(* Logix 5000 project; controller HP_SSC01 vendor 1 type 14 code 67 rev 17.7; software revision 17.01; part 9 of 15 *)
(* tags used below, declared in another part *)
   A_C3_0218 : ALIAS FOR S_C3_FaultSafety.18;
   A_C3_0219 : ALIAS FOR S_C3_FaultSafety.19;
   A_C3_0220 : ALIAS FOR S_C3_FaultSafety.20;
   A_C3_0221 : ALIAS FOR S_C3_FaultSafety.21;
   A_C3_0222 : ALIAS FOR S_C3_FaultSafety.22;
   A_C3_0223 : ALIAS FOR S_C3_FaultSafety.23;
   A_C3_0311 : ALIAS FOR C3_FaultStandard.11;
   A_C3_0312 : ALIAS FOR C3_FaultStandard.12;
   A_C3_0313 : ALIAS FOR C3_FaultStandard.13;
   A_C3_0314 : ALIAS FOR C3_FaultStandard.14;
   A_C3_0315 : ALIAS FOR C3_FaultStandard.15;
   C3 : AXIS_SERVO_DRIVE;
   C3_EncoderDegree : REAL;
   C3_EncoderPositionAtHome : DINT;
   C3_ExcecutePBHoldTimer : TIMER;
   C3_FaultHomeSwitchNotFound : BOOL;
   C3_Homed : BOOL;
   C3_HomeDelay : TIMER[8];
   C3_HomeFindSwitchMAM01 : MOTION_INSTRUCTION;
   C3_HomeFindSwitchMAM02 : MOTION_INSTRUCTION;
   C3_HomeFindSwitchMAS01 : MOTION_INSTRUCTION;
   C3_HomeGetCloseToSwitchMAM01 : MOTION_INSTRUCTION;
   C3_HomeGoToOnPathMAM01 : MOTION_INSTRUCTION;
   C3_HomeMessageNumber : DINT;
   C3_HomeSensorTestMAM02 : MOTION_INSTRUCTION;
   C3_HomeSequence : DINT;
   C3_HomeSequenceAlarms : DINT;
   C3_HomeSequenceAlarmTimer : TIMER[32];
   C3_HomeSequenceInProcess : BOOL;
   C3_HomeSequenceMAH : MOTION_INSTRUCTION;
   C3_HomeSwitchFaultK7KFailedOff : BOOL;
   C3_HomeSwitchFaultK7KFailedOn : BOOL;
   C3_HomeSwitchFaultSafeFailedOff : BOOL;
   C3_HomeSwitchFaultSafeFailedOn : BOOL;
   C3_HomeTest : REAL;
   C3_IndexEnable : BOOL;
   C3_IndexEnableTOF : TIMER;
   C3_IndexMAM01 : MOTION_INSTRUCTION;
   C3_IndexMAS01 : MOTION_INSTRUCTION;
   C3_IndexMessageNumber : DINT;
   C3_IndexPermissive : BOOL;
   C3_Jog_ONS : DINT;
   C3_JogDirection : DINT;
   C3_JogEnable : BOOL;
   C3_JogEnableTOF : TIMER;
   C3_JogForwardFastSelected : BOOL;
   C3_JogForwardSlowSelected : BOOL;
   C3_JogMAJ01 : MOTION_INSTRUCTION;
   C3_JogMAJ02 : MOTION_INSTRUCTION;
   C3_JogMAS01 : MOTION_INSTRUCTION;
   C3_JogMessageNumber : DINT;
   C3_JogPermissive : BOOL;
   C3_JogReverseFastSelected : BOOL;
   C3_JogReverseSlowSelected : BOOL;
   C3_MAJAcceleration : REAL;
   C3_MAJDeceleration : REAL;
   C3_MAJSpeed : REAL;
   C3_OIT_Current : DINT;
   C3_RemoteHomeCMD : BOOL;
   C3_ServoActionStatusOnDelay : TIMER;
   C3_SetEncoderHomePosition : BOOL;
   C3HomeSensorTestMAM01 : MOTION_INSTRUCTION;
   C3HomeSequenceONS : BOOL;
   C3HomeSequenceONS2 : BOOL;
   S_C3_EncoderPositionAtHomeSet : BOOL;
   S_C3_ExecutePB : BOOL;
   S_C3_FaultReset : BOOL;
   S_C3_HomeSafePE : ALIAS FOR C3_Safe:I.Pt04Data;
   S_C3_ModeLocal : BOOL;
   S_C3_ModeRemote : BOOL;
   S_C3_MSTOP_InputOK : BOOL;
   S_EncoderCtsFor360Deg : DINT;
(* Carousel3, continued *)

ROUTINE C330_Home   (* ladder *)
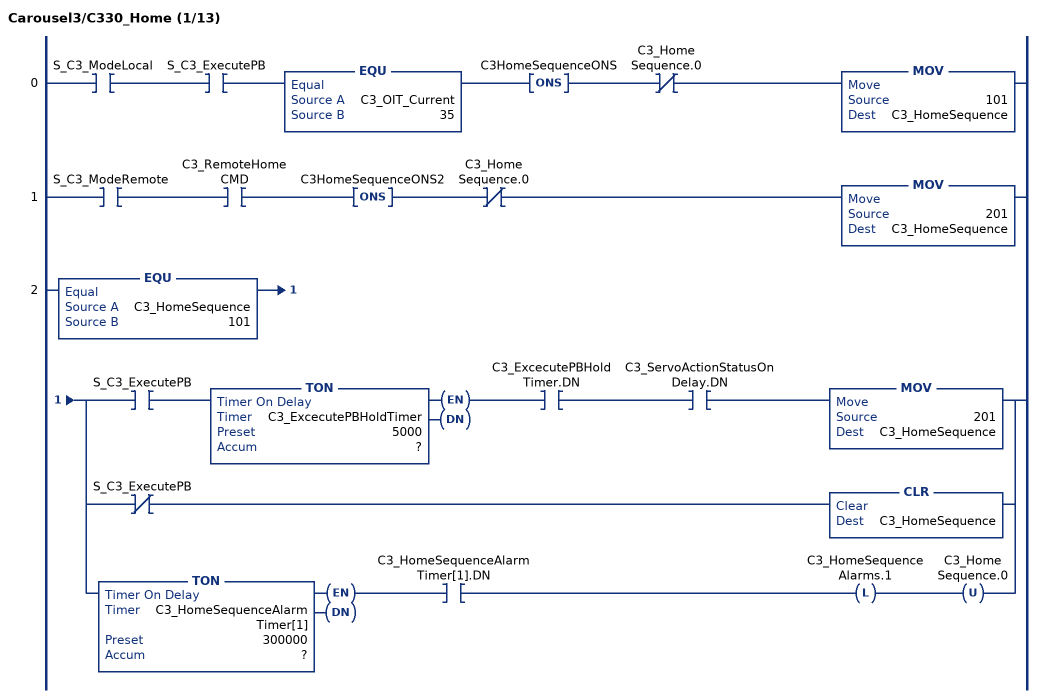
   0: XIC(S_C3_ModeLocal)XIC(S_C3_ExecutePB)EQU(C3_OIT_Current,35)ONS(C3HomeSequenceONS)XIO(C3_HomeSequence.0)MOV(101,C3_HomeSequence);
   1: XIC(S_C3_ModeRemote)XIC(C3_RemoteHomeCMD)ONS(C3HomeSequenceONS2)XIO(C3_HomeSequence.0)MOV(201,C3_HomeSequence);
   2: EQU(C3_HomeSequence,101)[XIC(S_C3_ExecutePB) TON(C3_ExcecutePBHoldTimer,?,?) XIC(C3_ExcecutePBHoldTimer.DN) XIC(C3_ServoActionStatusOnDelay.DN) MOV(201,C3_HomeSequence) ,XIO(S_C3_ExecutePB) CLR(C3_HomeSequence) ,TON(C3_HomeSequenceAlarmTimer[1],?,?) XIC(C3_HomeSequenceAlarmTimer[1].DN) OTL(C3_HomeSequenceAlarms.1) OTU(C3_HomeSequence.0) ];
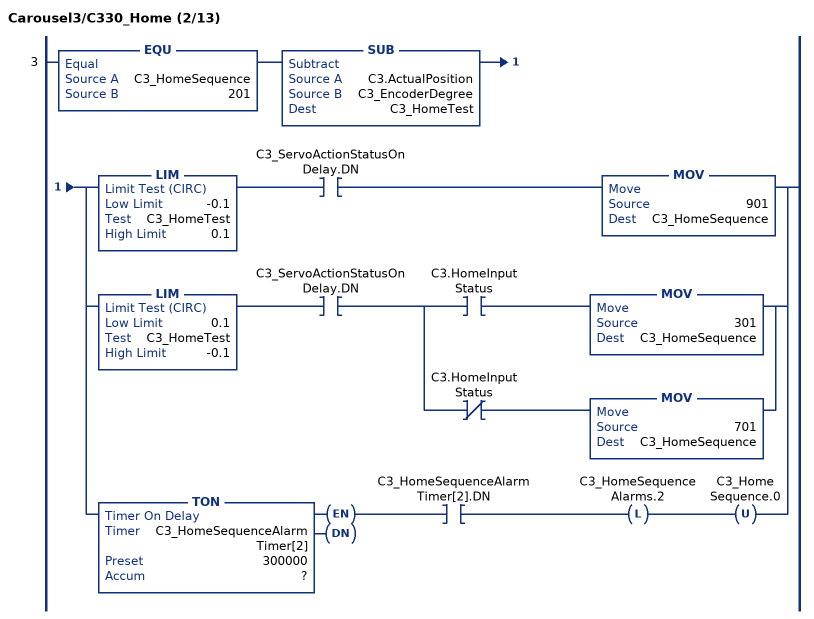
   3: EQU(C3_HomeSequence,201)SUB(C3.ActualPosition,C3_EncoderDegree,C3_HomeTest)[LIM(-0.1,C3_HomeTest,0.1) XIC(C3_ServoActionStatusOnDelay.DN) MOV(901,C3_HomeSequence) ,LIM(0.1,C3_HomeTest,-0.1) XIC(C3_ServoActionStatusOnDelay.DN) [XIC(C3.HomeInputStatus) MOV(301,C3_HomeSequence) ,XIO(C3.HomeInputStatus) MOV(701,C3_HomeSequence) ] ,TON(C3_HomeSequenceAlarmTimer[2],?,?) XIC(C3_HomeSequenceAlarmTimer[2].DN) OTL(C3_HomeSequenceAlarms.2) OTU(C3_HomeSequence.0) ];
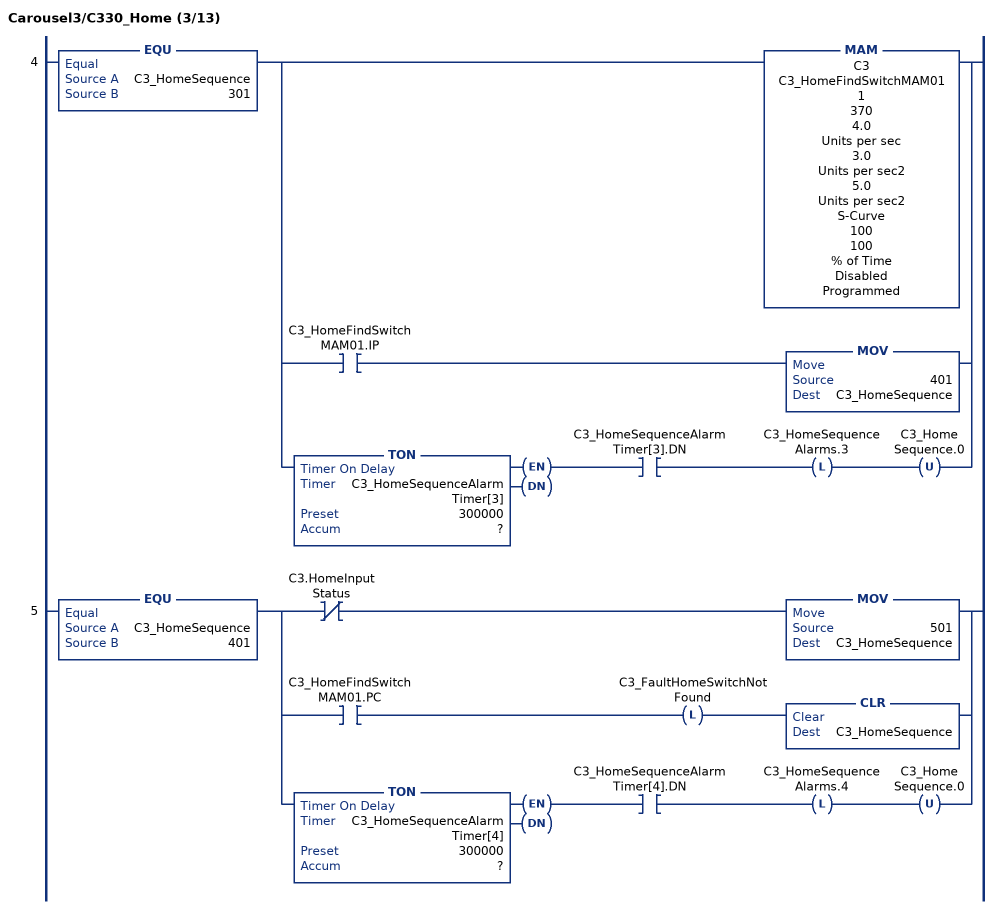
   4: EQU(C3_HomeSequence,301)[MAM(C3,C3_HomeFindSwitchMAM01,1,370,4.0,Units per sec,3.0,Units per sec2,5.0,Units per sec2,S-Curve,100,100,% of Time,Disabled,Programmed) ,XIC(C3_HomeFindSwitchMAM01.IP) MOV(401,C3_HomeSequence) ,TON(C3_HomeSequenceAlarmTimer[3],?,?) XIC(C3_HomeSequenceAlarmTimer[3].DN) OTL(C3_HomeSequenceAlarms.3) OTU(C3_HomeSequence.0) ];
   5: EQU(C3_HomeSequence,401)[XIO(C3.HomeInputStatus) MOV(501,C3_HomeSequence) ,XIC(C3_HomeFindSwitchMAM01.PC) OTL(C3_FaultHomeSwitchNotFound) CLR(C3_HomeSequence) ,TON(C3_HomeSequenceAlarmTimer[4],?,?) XIC(C3_HomeSequenceAlarmTimer[4].DN) OTL(C3_HomeSequenceAlarms.4) OTU(C3_HomeSequence.0) ];
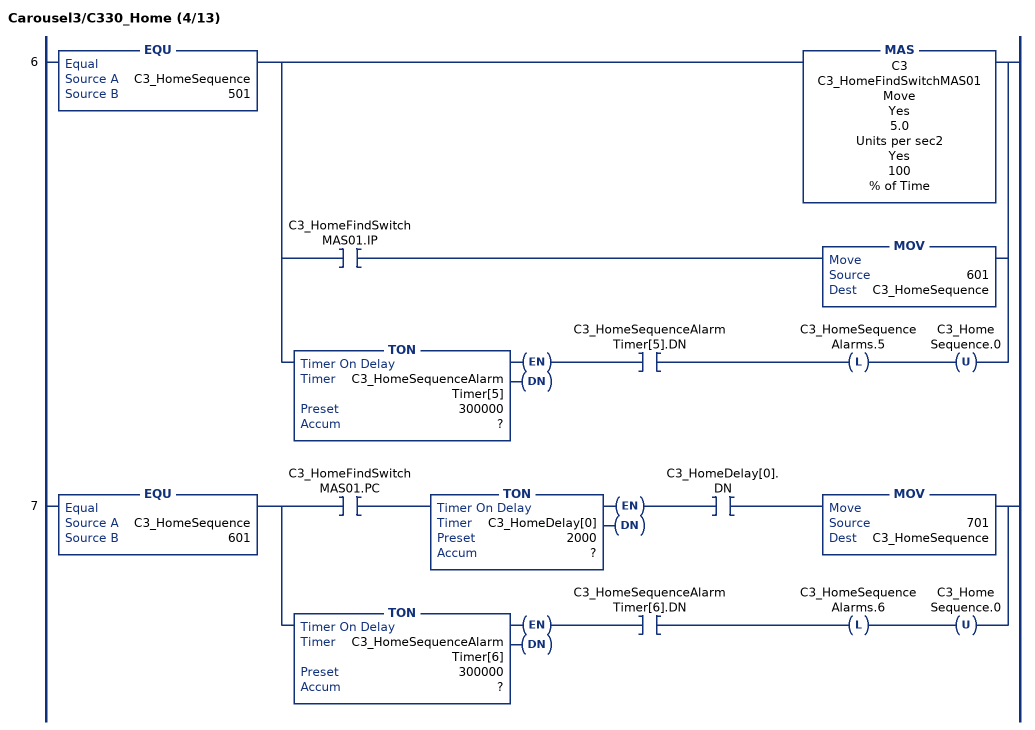
   6: EQU(C3_HomeSequence,501)[MAS(C3,C3_HomeFindSwitchMAS01,Move,Yes,5.0,Units per sec2,Yes,100,% of Time) ,XIC(C3_HomeFindSwitchMAS01.IP) MOV(601,C3_HomeSequence) ,TON(C3_HomeSequenceAlarmTimer[5],?,?) XIC(C3_HomeSequenceAlarmTimer[5].DN) OTL(C3_HomeSequenceAlarms.5) OTU(C3_HomeSequence.0) ];
   7: EQU(C3_HomeSequence,601)[XIC(C3_HomeFindSwitchMAS01.PC) TON(C3_HomeDelay[0],?,?) XIC(C3_HomeDelay[0].DN) MOV(701,C3_HomeSequence) ,TON(C3_HomeSequenceAlarmTimer[6],?,?) XIC(C3_HomeSequenceAlarmTimer[6].DN) OTL(C3_HomeSequenceAlarms.6) OTU(C3_HomeSequence.0) ];
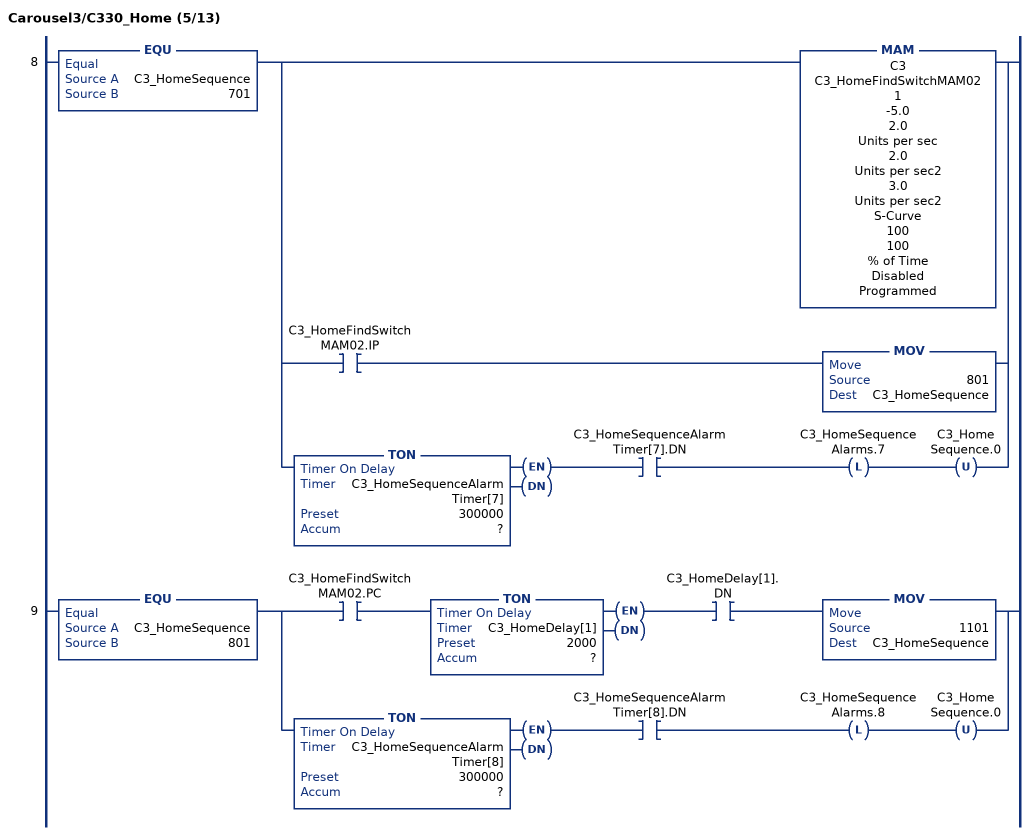
   8: EQU(C3_HomeSequence,701)[MAM(C3,C3_HomeFindSwitchMAM02,1,-5.0,2.0,Units per sec,2.0,Units per sec2,3.0,Units per sec2,S-Curve,100,100,% of Time,Disabled,Programmed) ,XIC(C3_HomeFindSwitchMAM02.IP) MOV(801,C3_HomeSequence) ,TON(C3_HomeSequenceAlarmTimer[7],?,?) XIC(C3_HomeSequenceAlarmTimer[7].DN) OTL(C3_HomeSequenceAlarms.7) OTU(C3_HomeSequence.0) ];
   9: EQU(C3_HomeSequence,801)[XIC(C3_HomeFindSwitchMAM02.PC) TON(C3_HomeDelay[1],?,?) XIC(C3_HomeDelay[1].DN) MOV(1101,C3_HomeSequence) ,TON(C3_HomeSequenceAlarmTimer[8],?,?) XIC(C3_HomeSequenceAlarmTimer[8].DN) OTL(C3_HomeSequenceAlarms.8) OTU(C3_HomeSequence.0) ];
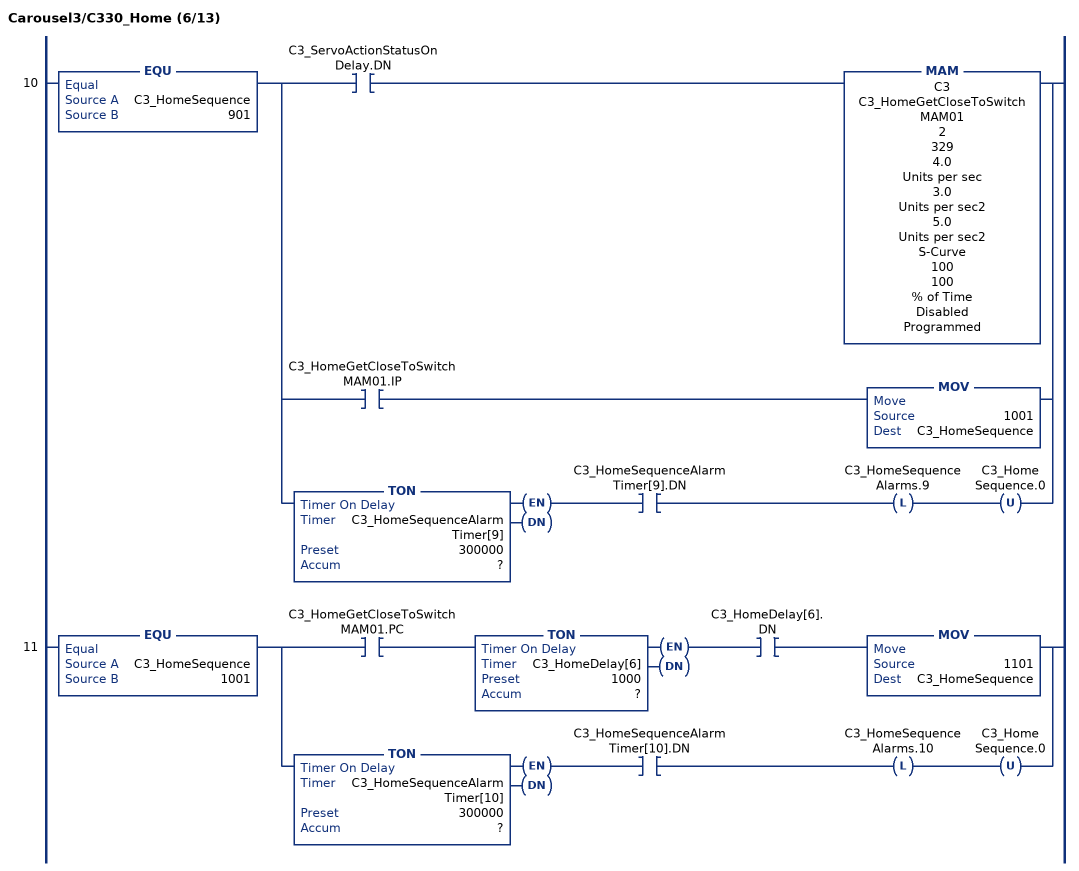
   10: EQU(C3_HomeSequence,901)[XIC(C3_ServoActionStatusOnDelay.DN) MAM(C3,C3_HomeGetCloseToSwitchMAM01,2,329,4.0,Units per sec,3.0,Units per sec2,5.0,Units per sec2,S-Curve,100,100,% of Time,Disabled,Programmed) ,XIC(C3_HomeGetCloseToSwitchMAM01.IP) MOV(1001,C3_HomeSequence) ,TON(C3_HomeSequenceAlarmTimer[9],?,?) XIC(C3_HomeSequenceAlarmTimer[9].DN) OTL(C3_HomeSequenceAlarms.9) OTU(C3_HomeSequence.0) ];
   11: EQU(C3_HomeSequence,1001)[XIC(C3_HomeGetCloseToSwitchMAM01.PC) TON(C3_HomeDelay[6],?,?) XIC(C3_HomeDelay[6].DN) MOV(1101,C3_HomeSequence) ,TON(C3_HomeSequenceAlarmTimer[10],?,?) XIC(C3_HomeSequenceAlarmTimer[10].DN) OTL(C3_HomeSequenceAlarms.10) OTU(C3_HomeSequence.0) ];
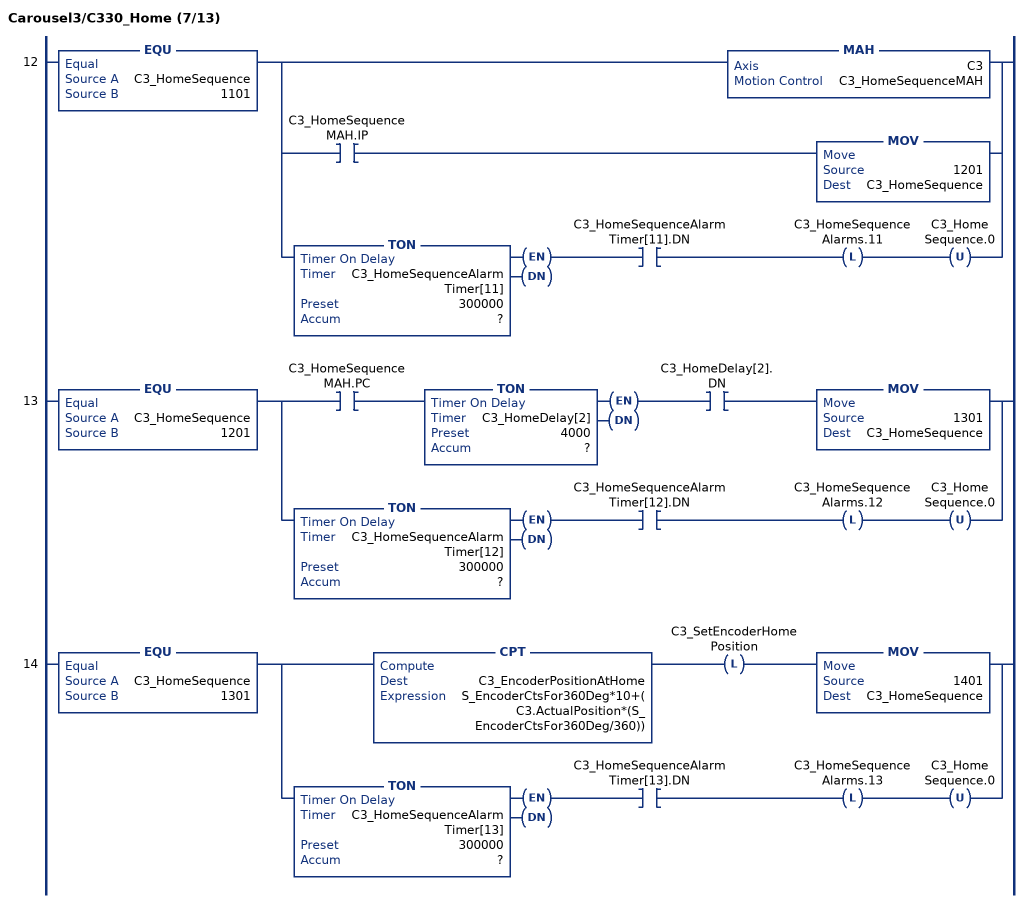
   12: EQU(C3_HomeSequence,1101)[MAH(C3,C3_HomeSequenceMAH) ,XIC(C3_HomeSequenceMAH.IP) MOV(1201,C3_HomeSequence) ,TON(C3_HomeSequenceAlarmTimer[11],?,?) XIC(C3_HomeSequenceAlarmTimer[11].DN) OTL(C3_HomeSequenceAlarms.11) OTU(C3_HomeSequence.0) ];
   13: EQU(C3_HomeSequence,1201)[XIC(C3_HomeSequenceMAH.PC) TON(C3_HomeDelay[2],?,?) XIC(C3_HomeDelay[2].DN) MOV(1301,C3_HomeSequence) ,TON(C3_HomeSequenceAlarmTimer[12],?,?) XIC(C3_HomeSequenceAlarmTimer[12].DN) OTL(C3_HomeSequenceAlarms.12) OTU(C3_HomeSequence.0) ];
   14: EQU(C3_HomeSequence,1301)[CPT(C3_EncoderPositionAtHome,S_EncoderCtsFor360Deg*10+(C3.ActualPosition*(S_EncoderCtsFor360Deg/360))) OTL(C3_SetEncoderHomePosition) MOV(1401,C3_HomeSequence) ,TON(C3_HomeSequenceAlarmTimer[13],?,?) XIC(C3_HomeSequenceAlarmTimer[13].DN) OTL(C3_HomeSequenceAlarms.13) OTU(C3_HomeSequence.0) ];
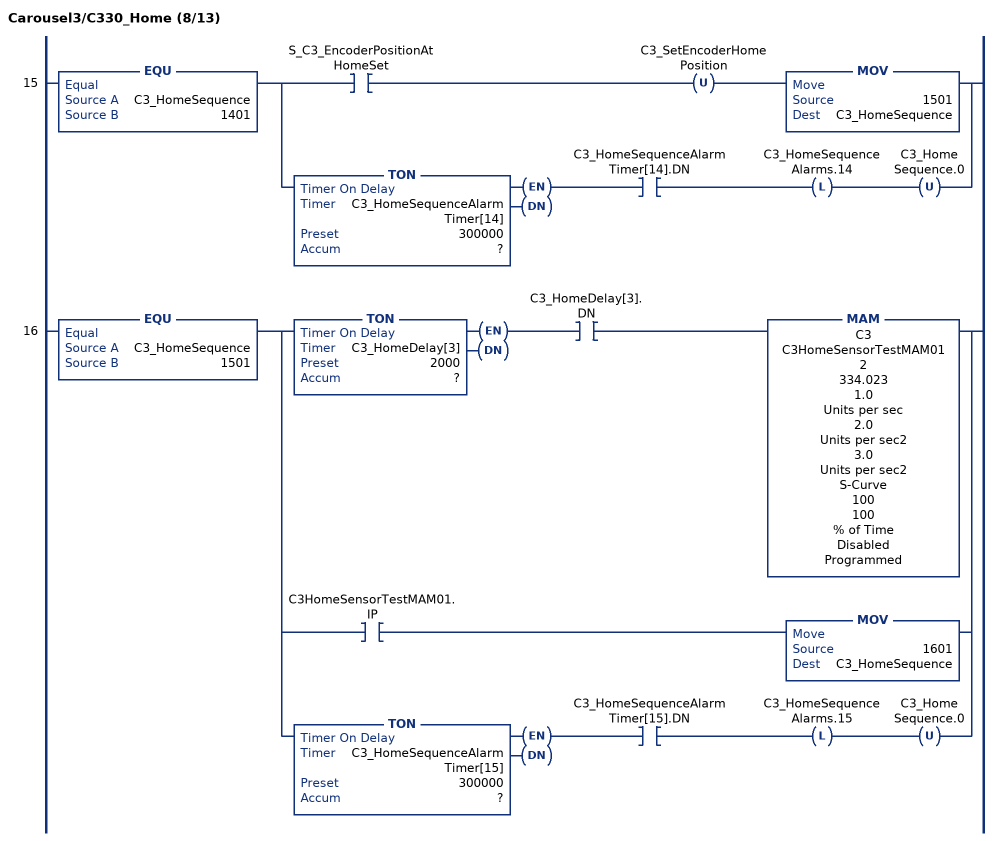
   15: EQU(C3_HomeSequence,1401)[XIC(S_C3_EncoderPositionAtHomeSet) OTU(C3_SetEncoderHomePosition) MOV(1501,C3_HomeSequence) ,TON(C3_HomeSequenceAlarmTimer[14],?,?) XIC(C3_HomeSequenceAlarmTimer[14].DN) OTL(C3_HomeSequenceAlarms.14) OTU(C3_HomeSequence.0) ];
   16: EQU(C3_HomeSequence,1501)[TON(C3_HomeDelay[3],?,?) XIC(C3_HomeDelay[3].DN) MAM(C3,C3HomeSensorTestMAM01,2,334.023,1.0,Units per sec,2.0,Units per sec2,3.0,Units per sec2,S-Curve,100,100,% of Time,Disabled,Programmed) ,XIC(C3HomeSensorTestMAM01.IP) MOV(1601,C3_HomeSequence) ,TON(C3_HomeSequenceAlarmTimer[15],?,?) XIC(C3_HomeSequenceAlarmTimer[15].DN) OTL(C3_HomeSequenceAlarms.15) OTU(C3_HomeSequence.0) ];
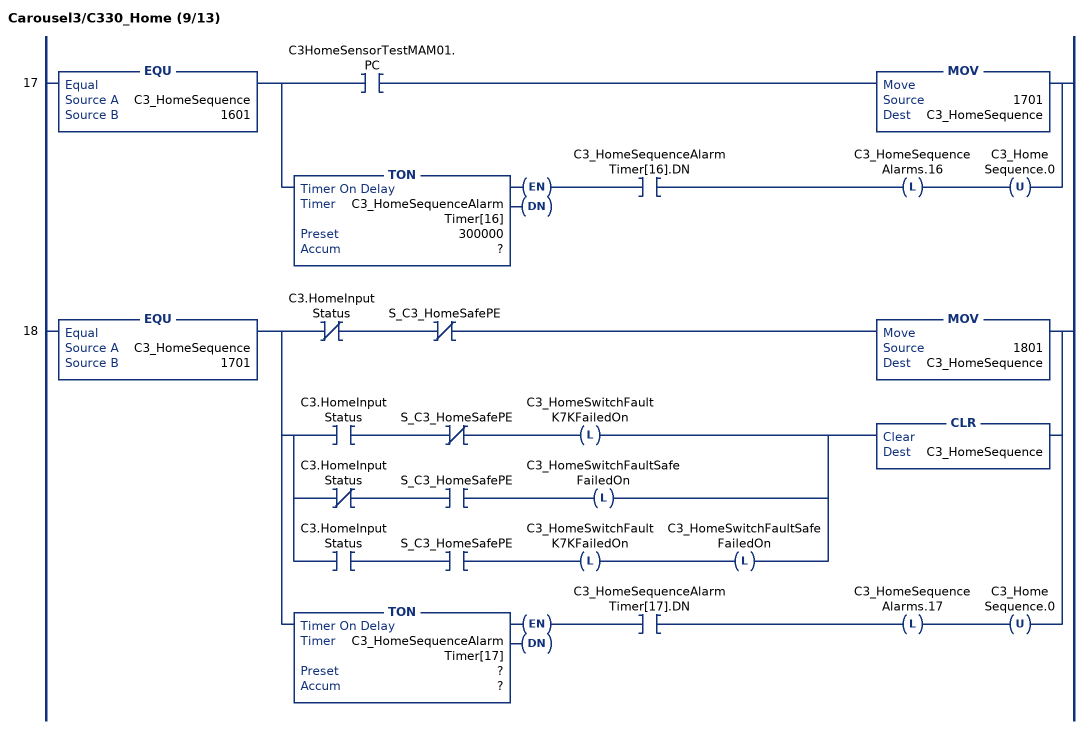
   17: EQU(C3_HomeSequence,1601)[XIC(C3HomeSensorTestMAM01.PC) MOV(1701,C3_HomeSequence) ,TON(C3_HomeSequenceAlarmTimer[16],?,?) XIC(C3_HomeSequenceAlarmTimer[16].DN) OTL(C3_HomeSequenceAlarms.16) OTU(C3_HomeSequence.0) ];
   18: EQU(C3_HomeSequence,1701)[XIO(C3.HomeInputStatus) XIO(S_C3_HomeSafePE) MOV(1801,C3_HomeSequence) ,[XIC(C3.HomeInputStatus) XIO(S_C3_HomeSafePE) OTL(C3_HomeSwitchFaultK7KFailedOn) ,XIO(C3.HomeInputStatus) XIC(S_C3_HomeSafePE) OTL(C3_HomeSwitchFaultSafeFailedOn) ,XIC(C3.HomeInputStatus) XIC(S_C3_HomeSafePE) OTL(C3_HomeSwitchFaultK7KFailedOn) OTL(C3_HomeSwitchFaultSafeFailedOn) ] CLR(C3_HomeSequence) ,TON(C3_HomeSequenceAlarmTimer[17],?,?) XIC(C3_HomeSequenceAlarmTimer[17].DN) OTL(C3_HomeSequenceAlarms.17) OTU(C3_HomeSequence.0) ];
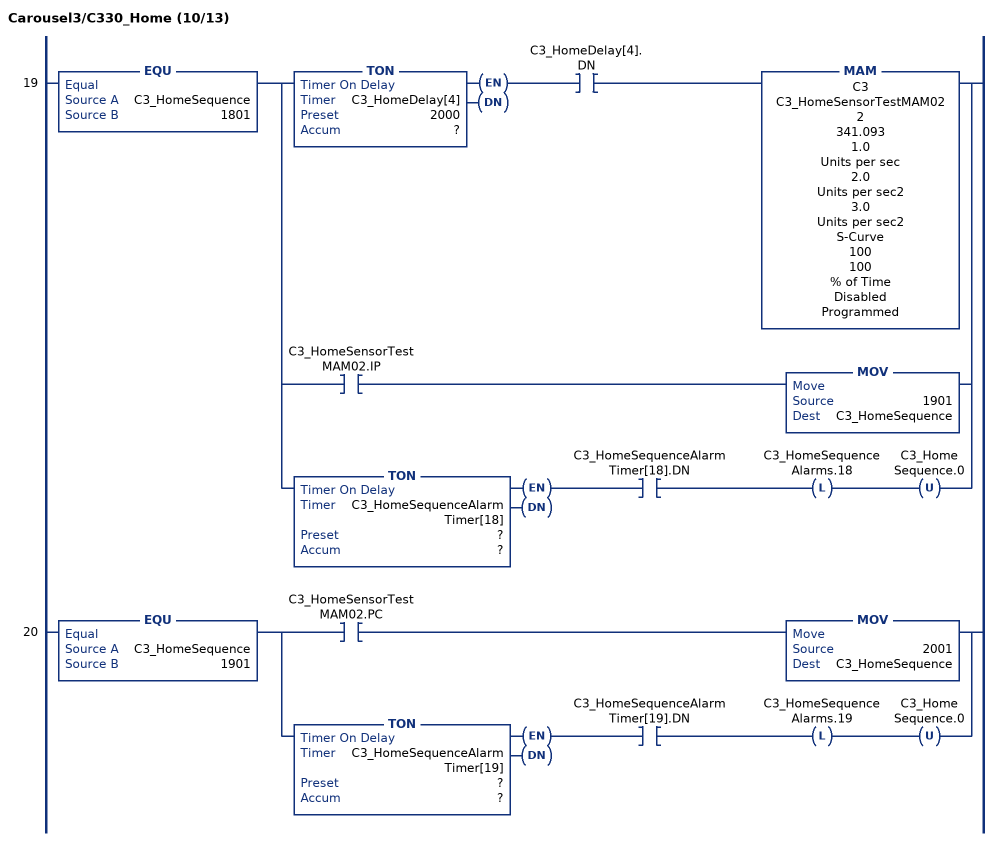
   19: EQU(C3_HomeSequence,1801)[TON(C3_HomeDelay[4],?,?) XIC(C3_HomeDelay[4].DN) MAM(C3,C3_HomeSensorTestMAM02,2,341.093,1.0,Units per sec,2.0,Units per sec2,3.0,Units per sec2,S-Curve,100,100,% of Time,Disabled,Programmed) ,XIC(C3_HomeSensorTestMAM02.IP) MOV(1901,C3_HomeSequence) ,TON(C3_HomeSequenceAlarmTimer[18],?,?) XIC(C3_HomeSequenceAlarmTimer[18].DN) OTL(C3_HomeSequenceAlarms.18) OTU(C3_HomeSequence.0) ];
   20: EQU(C3_HomeSequence,1901)[XIC(C3_HomeSensorTestMAM02.PC) MOV(2001,C3_HomeSequence) ,TON(C3_HomeSequenceAlarmTimer[19],?,?) XIC(C3_HomeSequenceAlarmTimer[19].DN) OTL(C3_HomeSequenceAlarms.19) OTU(C3_HomeSequence.0) ];
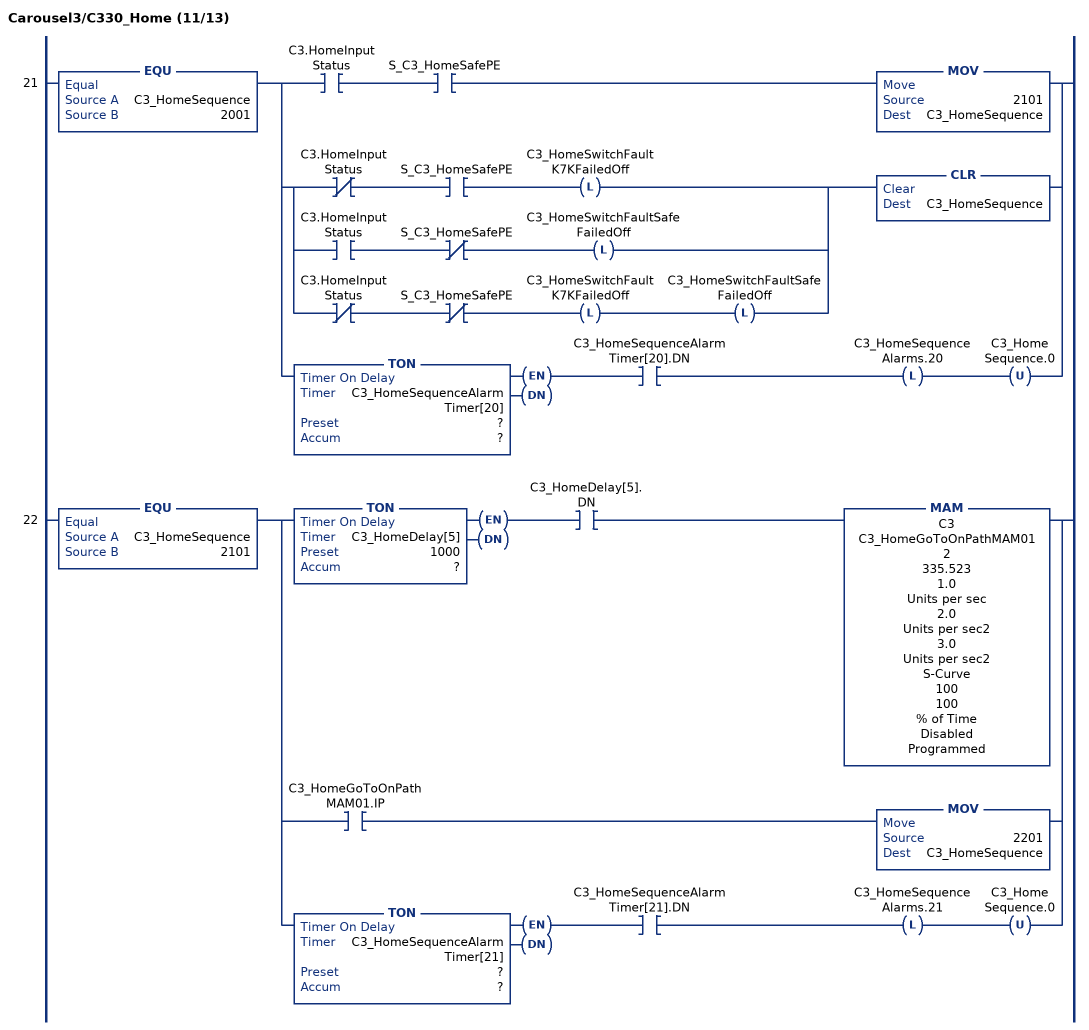
   21: EQU(C3_HomeSequence,2001)[XIC(C3.HomeInputStatus) XIC(S_C3_HomeSafePE) MOV(2101,C3_HomeSequence) ,[XIO(C3.HomeInputStatus) XIC(S_C3_HomeSafePE) OTL(C3_HomeSwitchFaultK7KFailedOff) ,XIC(C3.HomeInputStatus) XIO(S_C3_HomeSafePE) OTL(C3_HomeSwitchFaultSafeFailedOff) ,XIO(C3.HomeInputStatus) XIO(S_C3_HomeSafePE) OTL(C3_HomeSwitchFaultK7KFailedOff) OTL(C3_HomeSwitchFaultSafeFailedOff) ] CLR(C3_HomeSequence) ,TON(C3_HomeSequenceAlarmTimer[20],?,?) XIC(C3_HomeSequenceAlarmTimer[20].DN) OTL(C3_HomeSequenceAlarms.20) OTU(C3_HomeSequence.0) ];
   22: EQU(C3_HomeSequence,2101)[TON(C3_HomeDelay[5],?,?) XIC(C3_HomeDelay[5].DN) MAM(C3,C3_HomeGoToOnPathMAM01,2,335.523,1.0,Units per sec,2.0,Units per sec2,3.0,Units per sec2,S-Curve,100,100,% of Time,Disabled,Programmed) ,XIC(C3_HomeGoToOnPathMAM01.IP) MOV(2201,C3_HomeSequence) ,TON(C3_HomeSequenceAlarmTimer[21],?,?) XIC(C3_HomeSequenceAlarmTimer[21].DN) OTL(C3_HomeSequenceAlarms.21) OTU(C3_HomeSequence.0) ];
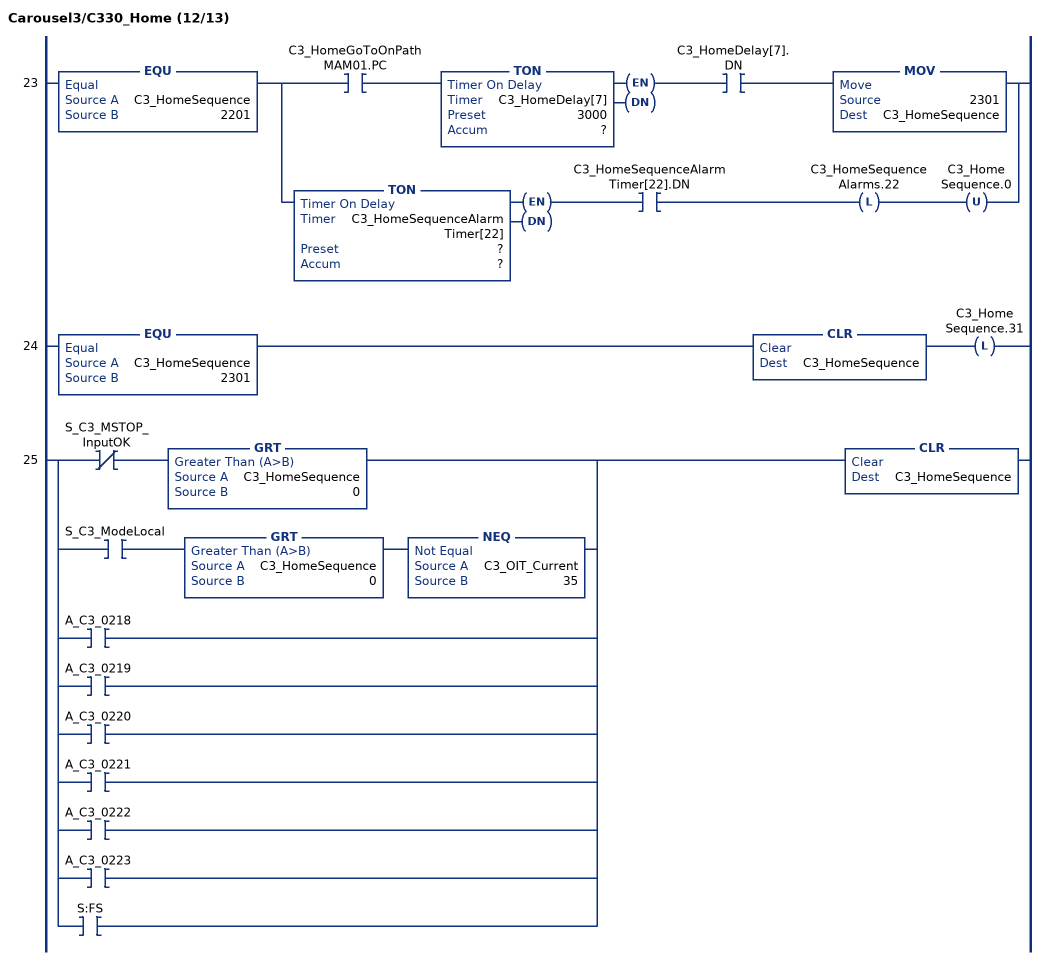
   23: EQU(C3_HomeSequence,2201)[XIC(C3_HomeGoToOnPathMAM01.PC) TON(C3_HomeDelay[7],?,?) XIC(C3_HomeDelay[7].DN) MOV(2301,C3_HomeSequence) ,TON(C3_HomeSequenceAlarmTimer[22],?,?) XIC(C3_HomeSequenceAlarmTimer[22].DN) OTL(C3_HomeSequenceAlarms.22) OTU(C3_HomeSequence.0) ];
   24: EQU(C3_HomeSequence,2301)CLR(C3_HomeSequence)OTL(C3_HomeSequence.31);
   25: [XIO(S_C3_MSTOP_InputOK) GRT(C3_HomeSequence,0) ,XIC(S_C3_ModeLocal) GRT(C3_HomeSequence,0) NEQ(C3_OIT_Current,35) ,XIC(A_C3_0218) ,XIC(A_C3_0219) ,XIC(A_C3_0220) ,XIC(A_C3_0221) ,XIC(A_C3_0222) ,XIC(A_C3_0223) ,XIC(S:FS) ]CLR(C3_HomeSequence);
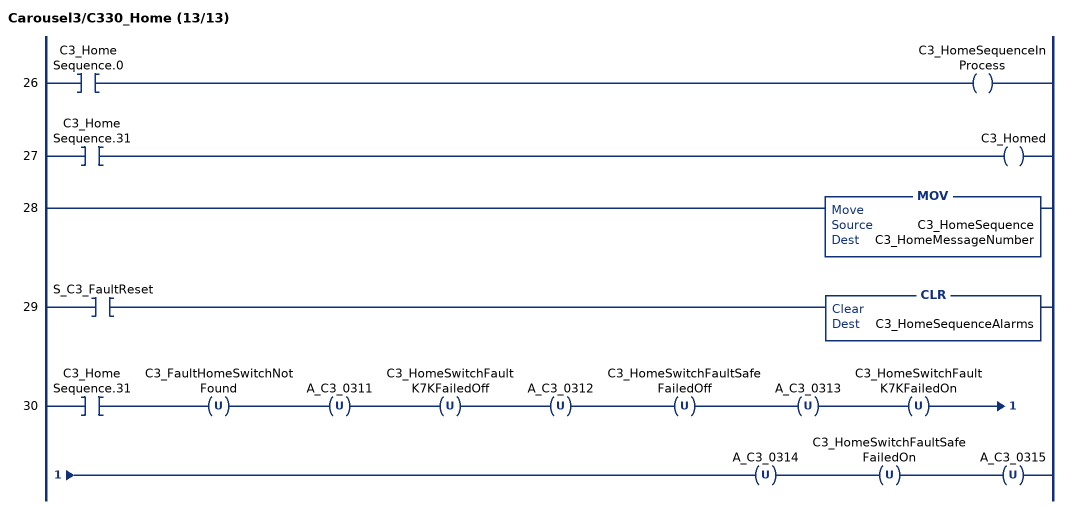
   26: XIC(C3_HomeSequence.0)OTE(C3_HomeSequenceInProcess);
   27: XIC(C3_HomeSequence.31)OTE(C3_Homed);
   28: MOV(C3_HomeSequence,C3_HomeMessageNumber);
   29: XIC(S_C3_FaultReset)CLR(C3_HomeSequenceAlarms);
   30: XIC(C3_HomeSequence.31)OTU(C3_FaultHomeSwitchNotFound)OTU(A_C3_0311)OTU(C3_HomeSwitchFaultK7KFailedOff)OTU(A_C3_0312)OTU(C3_HomeSwitchFaultSafeFailedOff)OTU(A_C3_0313)OTU(C3_HomeSwitchFaultK7KFailedOn)OTU(A_C3_0314)OTU(C3_HomeSwitchFaultSafeFailedOn)OTU(A_C3_0315);
END_ROUTINE

ROUTINE C335_Index   (* ladder *)
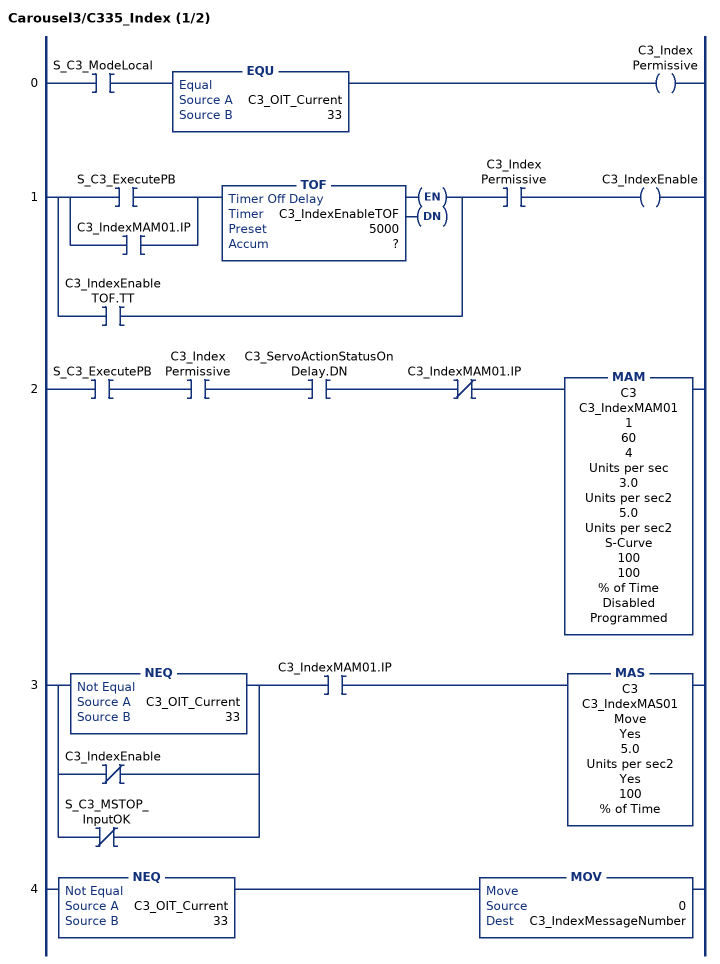
   0: XIC(S_C3_ModeLocal)EQU(C3_OIT_Current,33)OTE(C3_IndexPermissive);
   1: [[XIC(S_C3_ExecutePB) ,XIC(C3_IndexMAM01.IP) ] TOF(C3_IndexEnableTOF,?,?) ,XIC(C3_IndexEnableTOF.TT) ]XIC(C3_IndexPermissive)OTE(C3_IndexEnable);
   2: XIC(S_C3_ExecutePB)XIC(C3_IndexPermissive)XIC(C3_ServoActionStatusOnDelay.DN)XIO(C3_IndexMAM01.IP)MAM(C3,C3_IndexMAM01,1,60,4,Units per sec,3.0,Units per sec2,5.0,Units per sec2,S-Curve,100,100,% of Time,Disabled,Programmed);
   3: [NEQ(C3_OIT_Current,33) ,XIO(C3_IndexEnable) ,XIO(S_C3_MSTOP_InputOK) ]XIC(C3_IndexMAM01.IP)MAS(C3,C3_IndexMAS01,Move,Yes,5.0,Units per sec2,Yes,100,% of Time);
   4: NEQ(C3_OIT_Current,33)MOV(0,C3_IndexMessageNumber);
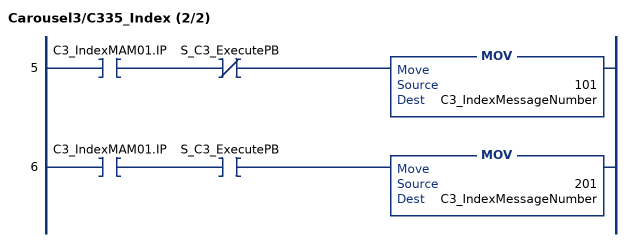
   5: XIC(C3_IndexMAM01.IP)XIO(S_C3_ExecutePB)MOV(101,C3_IndexMessageNumber);
   6: XIC(C3_IndexMAM01.IP)XIC(S_C3_ExecutePB)MOV(201,C3_IndexMessageNumber);
END_ROUTINE

ROUTINE C340_Jog   (* ladder *)
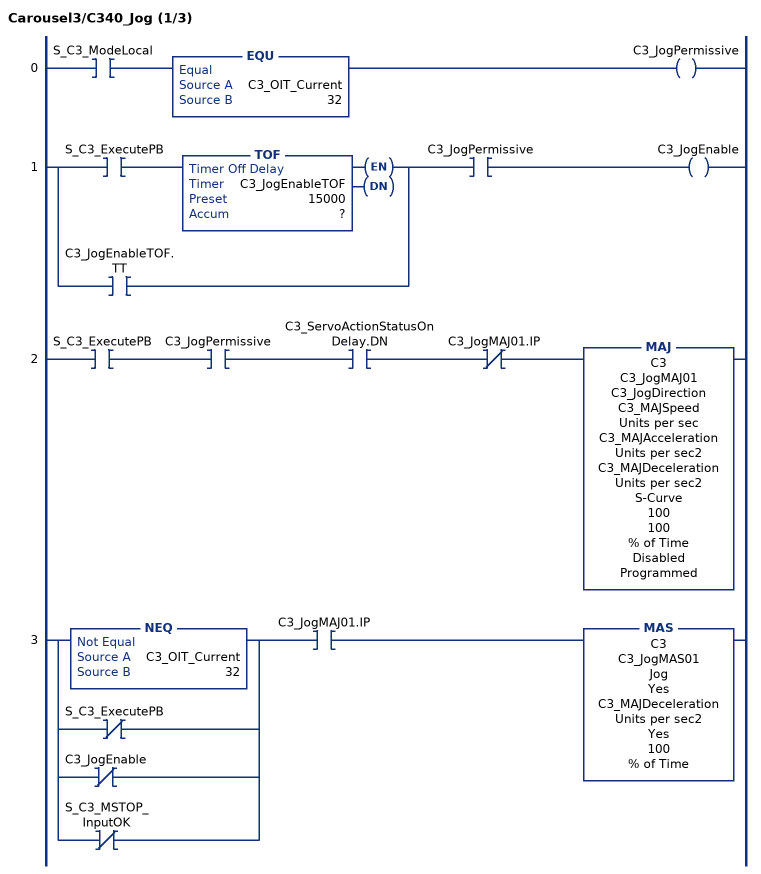
   0: XIC(S_C3_ModeLocal)EQU(C3_OIT_Current,32)OTE(C3_JogPermissive);
   1: [XIC(S_C3_ExecutePB) TOF(C3_JogEnableTOF,?,?) ,XIC(C3_JogEnableTOF.TT) ]XIC(C3_JogPermissive)OTE(C3_JogEnable);
   2: XIC(S_C3_ExecutePB)XIC(C3_JogPermissive)XIC(C3_ServoActionStatusOnDelay.DN)XIO(C3_JogMAJ01.IP)MAJ(C3,C3_JogMAJ01,C3_JogDirection,C3_MAJSpeed,Units per sec,C3_MAJAcceleration,Units per sec2,C3_MAJDeceleration,Units per sec2,S-Curve,100,100,% of Time,Disabled,Programmed);
   3: [NEQ(C3_OIT_Current,32) ,XIO(S_C3_ExecutePB) ,XIO(C3_JogEnable) ,XIO(S_C3_MSTOP_InputOK) ]XIC(C3_JogMAJ01.IP)MAS(C3,C3_JogMAS01,Jog,Yes,C3_MAJDeceleration,Units per sec2,Yes,100,% of Time);
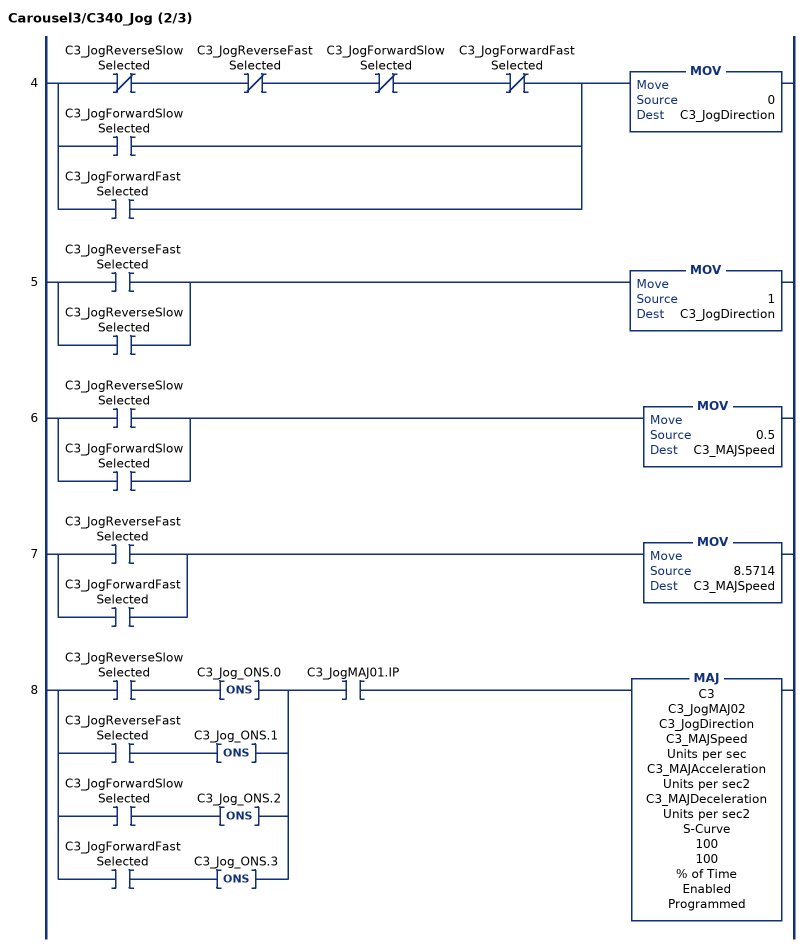
   4: [XIO(C3_JogReverseSlowSelected) XIO(C3_JogReverseFastSelected) XIO(C3_JogForwardSlowSelected) XIO(C3_JogForwardFastSelected) ,XIC(C3_JogForwardSlowSelected) ,XIC(C3_JogForwardFastSelected) ]MOV(0,C3_JogDirection);
   5: [XIC(C3_JogReverseFastSelected) ,XIC(C3_JogReverseSlowSelected) ]MOV(1,C3_JogDirection);
   6: [XIC(C3_JogReverseSlowSelected) ,XIC(C3_JogForwardSlowSelected) ]MOV(0.5,C3_MAJSpeed);
   7: [XIC(C3_JogReverseFastSelected) ,XIC(C3_JogForwardFastSelected) ]MOV(8.5714,C3_MAJSpeed);
   8: [XIC(C3_JogReverseSlowSelected) ONS(C3_Jog_ONS.0) ,XIC(C3_JogReverseFastSelected) ONS(C3_Jog_ONS.1) ,XIC(C3_JogForwardSlowSelected) ONS(C3_Jog_ONS.2) ,XIC(C3_JogForwardFastSelected) ONS(C3_Jog_ONS.3) ]XIC(C3_JogMAJ01.IP)MAJ(C3,C3_JogMAJ02,C3_JogDirection,C3_MAJSpeed,Units per sec,C3_MAJAcceleration,Units per sec2,C3_MAJDeceleration,Units per sec2,S-Curve,100,100,% of Time,Enabled,Programmed);
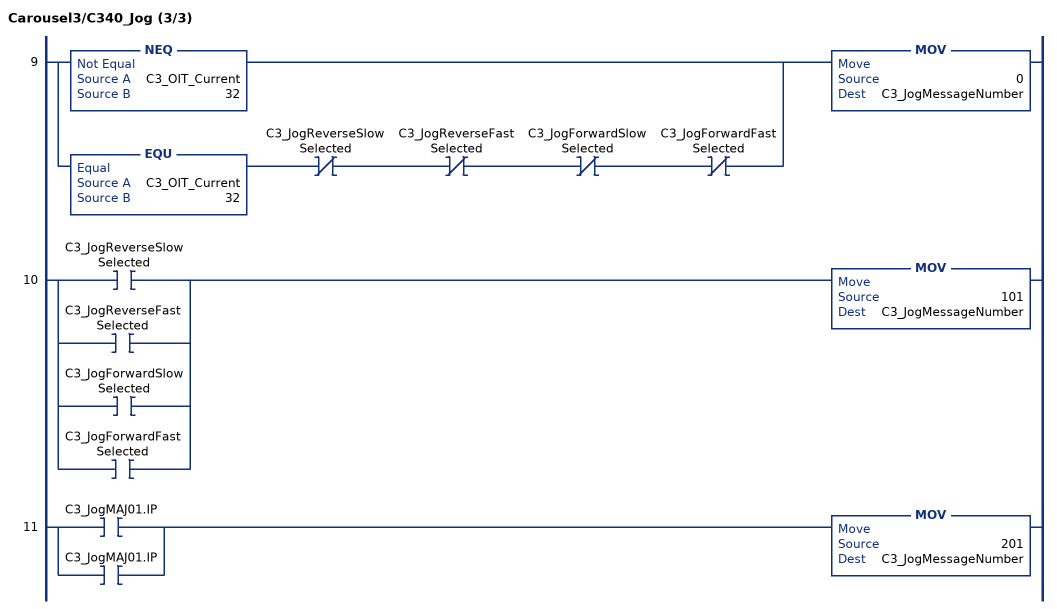
   9: [NEQ(C3_OIT_Current,32) ,EQU(C3_OIT_Current,32) XIO(C3_JogReverseSlowSelected) XIO(C3_JogReverseFastSelected) XIO(C3_JogForwardSlowSelected) XIO(C3_JogForwardFastSelected) ]MOV(0,C3_JogMessageNumber);
   10: [XIC(C3_JogReverseSlowSelected) ,XIC(C3_JogReverseFastSelected) ,XIC(C3_JogForwardSlowSelected) ,XIC(C3_JogForwardFastSelected) ]MOV(101,C3_JogMessageNumber);
   11: [XIC(C3_JogMAJ01.IP) ,XIC(C3_JogMAJ01.IP) ]MOV(201,C3_JogMessageNumber);
END_ROUTINE
